PROGRAM MAIN
VAR
	bTest: BOOL;
END_VAR

END_PROGRAM

(* stored: Version 1.1.0.1, ProductVersion 3.1.4024.12
   POU MAIN: Id {3af76850-7d8c-4443-bc25-119f4c03128e}, SpecialFunc None *)
